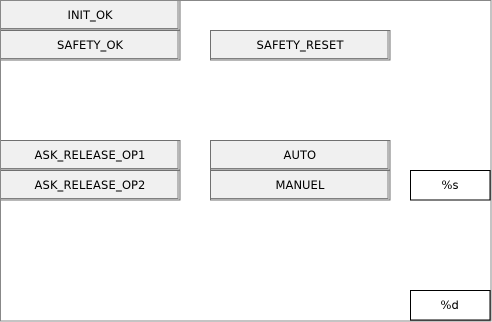
VISUALIZATION GEMMA  // 492x322
    Button (0,0 180x30), "INIT_OK", pressed state: Flag_Variables.FLAGS .INIT_OK
        toggle Flag_Variables.FLAGS .INIT_OK
    Button (0,30 180x30), "SAFETY_OK", pressed state: Flag_Variables.FLAGS .SAFETY_OK
        toggle Flag_Variables.FLAGS .SAFETY_OK
    Button (0,140 180x30), "ASK_RELEASE_OP1", pressed state: IOs_Variables.PRINT_DI .ASK_RELEASE_JIG_OP1
        toggle IOs_Variables.PRINT_DI .ASK_RELEASE_JIG_OP1
    Button (0,170 180x30), "ASK_RELEASE_OP2", pressed state: IOs_Variables.PRINT_DI .ASK_RELEASE_JIG_OP2
        toggle IOs_Variables.PRINT_DI .ASK_RELEASE_JIG_OP2
    Button (210,30 180x30), "SAFETY_RESET", pressed state: Flag_Variables.SAFETY_OUT .NOT_AUS_RESET
        toggle Flag_Variables.SAFETY_OUT .NOT_AUS_RESET
    Button (210,140 180x30), "AUTO", pressed state: Flag_Variables.FLAGS .AUTO
        toggle Flag_Variables.FLAGS .AUTO
    Button (210,170 180x30), "MANUEL", pressed state: Flag_Variables.FLAGS .MANUAL
        toggle Flag_Variables.FLAGS .MANUAL
    Rectangle (410,170 80x30), "%s", text variable: GEMMA.STEP
    Rectangle (410,290 80x30), "%d", text variable: LEDS.M1_FB_GetPositionIs.PositionIs
END_VISUALIZATION

(* stored: Version 1.1.0.1, ProductVersion 3.1.0.26
   Visu GEMMA: Id {edf7e6be-272d-4427-af33-c3435180b2af} *)
